FUNCTION FUN_ComputeMovingSetPoint_1 : REAL
VAR_INPUT
	currentTemp 		: REAL;
	targetSetPoint 		: REAL;
END_VAR	
VAR
	deltaTemp 			: REAL;
	sign				: REAL;
	maxDeltaTemp		: REAL;
END_VAR

deltaTemp := targetSetPoint - currentTemp;
maxDeltaTemp := 10.0;

IF deltaTemp >= 0 THEN
	sign := 1.0;
ELSE
	sign := -1.0;
END_IF

IF ABS(deltaTemp) > maxDeltaTemp THEN
	FUN_ComputeMovingSetPoint := sign*maxDeltaTemp + currentTemp;
ELSE
	FUN_ComputeMovingSetPoint := targetSetPoint;
END_IF

END_FUNCTION

(* stored: Version 1.1.0.1, ProductVersion 3.1.4022.12
   POU FUN_ComputeMovingSetPoint_1: Id {c3a9347f-eff5-4db1-b423-881656562795}, SpecialFunc None *)
